FUNCTION_BLOCK ExtractAirControl
VAR_INPUT
	EN: BOOL;
END_VAR
VAR_OUTPUT
	ENO: BOOL;
END_VAR
VAR
END_VAR

ENO := EN;

END_FUNCTION_BLOCK

(* stored: Version 1.1.0.1, ProductVersion 3.1.4024.3
   POU ExtractAirControl: Id {d099ca57-54fe-4b3f-a235-288be625a22c}, SpecialFunc None *)
